{attribute 'enable_dynamic_creation'}
FUNCTION_BLOCK FutureMCStop EXTENDS FB_AbstructFuture
VAR_INPUT
END_VAR
VAR_OUTPUT
END_VAR
VAR
	_axis: REFERENCE TO AXIS_REF;
	_mc_stop	: MC_Stop;
	_mc_reset	: MC_Reset;
	_deceleration: MC_LREAL;
	_jerk		: MC_LREAL;
	_option : ST_MoveOptions;
	_exec_state : UDINT;
END_VAR

METHOD error_reset : BOOL // Must be overrided if future has any errors.
IF _error_id <> 0 THEN
	CASE _exec_state OF
		0:
			_mc_reset(Axis := _axis, Execute := FALSE);
			_mc_reset(Axis:= _axis, Execute := TRUE );
			_exec_state := 1;
		1:
			IF _mc_reset.Busy THEN
				_mc_reset(Axis:= _axis,Execute := FALSE);
			END_IF
	END_CASE
	
	_error_id := _mc_reset.ErrorID;
	error_reset := _mc_reset.Done;
ELSE
	error_reset := TRUE;
END_IF
END_METHOD

METHOD execute : BOOL // Return TRUE if finish.

CASE _exec_state OF
	0:
		_mc_stop(axis := _axis, Execute := FALSE);
		_mc_stop(
			Axis:= _axis,
			Execute := TRUE,
			Jerk := _jerk,
			Options := _option
		);
		_exec_state := 1;
	1:
		IF _mc_stop.Busy THEN
			_mc_stop(Axis:= _axis,Execute := FALSE);
		END_IF
END_CASE

_error_id := _mc_stop.ErrorID;
execute := _mc_stop.Done OR _mc_stop.Error;
END_METHOD

METHOD init : BOOL // Return TRUE if finish.
_exec_state := 0;
init := TRUE;
END_METHOD

METHOD set_options : BOOL
VAR_INPUT
	option : ST_MoveOptions;
END_VAR
_option := option;
END_METHOD

METHOD set_parameters : BOOL
VAR_INPUT
	axis : REFERENCE TO AXIS_REF;
	deceleration	: MC_LREAL;		// Set deceleration in case let moving axis halt.
	jerk			: MC_LREAL;		// Set jerk in case let moving axis halt.
END_VAR
_axis REF= axis;
_deceleration := deceleration;
_jerk := jerk;
END_METHOD

END_FUNCTION_BLOCK

(* stored: Version 1.1.0.1, ProductVersion 3.1.4026.13
   POU FutureMCStop: Id {26698a42-81bf-4866-be85-711032f5993e}, SpecialFunc None
   Method error_reset: Id {b90342f2-8d7c-4ca3-8a9b-2fde84fe5763}
   Method execute: Id {5489d85d-357c-45ed-aba8-a7ed50652b80}
   Method init: Id {195059ec-0713-4e59-80cc-d37c784c8773}
   Method set_options: Id {d5b82e0f-9855-4e24-94e5-fe17a38beff1}
   Method set_parameters: Id {c2ef947b-5f79-4104-ada4-d1f1274db3dd} *)
